// TIA Portal V17 export
// export: Created 2025-03-07T09:19:57.2846838Z, ExportSetting WithDefaults, DisplayName Totally Integrated Automation Portal, DisplayVersion V17 Update 8, DisplayName TIA Portal Openness, DisplayVersion V17 Update 8, DisplayName TIA Portal Version Control Interface, DisplayVersion V17, DisplayName SINAMICS Startdrive Advanced, DisplayVersion V17 SP2, DisplayName SINAMICS Startdrive G110M, G120, G120C, G120D, G120P, G115D, DisplayVersion V17 SP2, DisplayName SINAMICS Startdrive G130, G150, S120, S150, SINAMICS MV, S210, DisplayVersion V17 SP2, DisplayName STEP 7 Professional, DisplayVersion V17 Update 8, DisplayName SINUMERIK ONE STEP 7 Toolbox, DisplayVersion V17 Update 12, DisplayName SINUMERIK 840D sl STEP 7 Toolbox, DisplayVersion V17 Update 12, DisplayName STEP 7 Safety, DisplayVersion V17 Update 6, DisplayName WinCC Advanced, DisplayVersion V17 Update 8
TYPE "LASER READY"
// stored: IsFailsafeCompliant false
   STRUCT
      "LASER READY LASER ARM INPUT ACKNOWLEDGE_1" : Bool;
      "LASER READY INPUT LASER EMERGENCY STOP" : Bool;
      "LASER READY INPUT LASER SC STATUS" : Bool;
      "LASER READY CIRCUIT BREAKER" : Bool;
      "LASER READY" : Bool;
      "LASER READY START GENERAL CONDITIONS" : Bool;
      "LASER READY START INITIAL CONDITIONS" : Bool;
      "LASER READY MANUAL START REQUEST" : Bool;
      "LASER READY AUTO START REQUEST" : Bool;
      "LASER READY START REQUEST" : Bool;
      "LASER READY START COMMAND" : Bool;
      "LASER READY LASER SYSTEM ON" : Bool;
      "LASER READY FEEDBACK ON" : Bool;
      "LASSER ANALOG CONTROL ACTIVE" : Bool;
      "LASER READY STOP GENERAL CONDITIONS" : Bool;
      "LASER READY STOP INITIAL CONDITIONS" : Bool;
      "LASER READY MANUAL STOP REQUEST" : Bool;
      "LASER READY AUTO STOP REQUEST" : Bool;
      "LASER READY STOP REQUEST" : Bool;
      "LASER READY STOP COMMAND" : Bool;
      "LASER READY STOPPED" : Bool;
      "LASER READY FEEDBACK OFF" : Bool;
      "LASER READY CIRCUIT BREAKER ALARM" : Bool;
      "LASER READY LASER ERROR" : Bool;
      "LASER READY WARNING LASER" : Bool;
      "LASER READY LASER NOT READY" : Bool;
      "LASER READY LASER NOT SWITCHED ON" : Bool;
      "LASER READY FAULT" : Bool;
      "LASER READY WARNING GONE" : Bool;
      "LASER READY START GENERAL CONDITION HELP" : Bool;
      "LASER READY START INITIAL CONDITION HELP" : Bool;
      "LASER READY STOP GENERAL CONDITION HELP" : Bool;
      "LASER READY STOP INITIAL CONDITION HELP" : Bool;
      "LASER MIN POWER LIMIT" : Int;
      "LASER MAX POWER LIMIT" : Int;
      "LASER POWER COMMAND" : Int;
      "TIMER AUTO REQ ON" : TON_TIME;
      "TIMER FAULT 1" { S7_SetPoint := 'True'} : TON_TIME;
      "TIMER FAULT 2" { S7_SetPoint := 'True'} : TON_TIME;
      "TIMER FAULT 3" { S7_SetPoint := 'True'} : TON_TIME;
      "TIMER LASER REQUEST" { S7_SetPoint := 'True'} : TON_TIME;
      "TIMER REST ERROR" { S7_SetPoint := 'True'} : TON_TIME;
   END_STRUCT;
END_TYPE
